// Mitsubishi GX Works2 project: questão_7   PLC: Q03UDV
// LRI_2023

PROGRAM MAIN
VAR
  yo : INT;
  TS0 : BOOL;
  RT0 : BOOL;
END_VAR
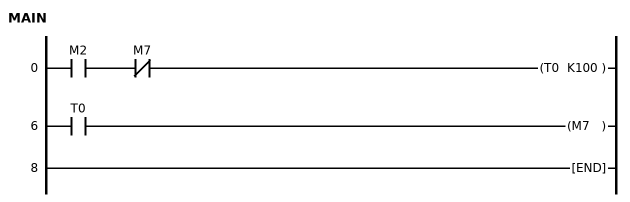
0     LD      M2
      ANI     M7
      OUT     T0 K100
6     LD      T0
      OUT     M7
8     END
END_PROGRAM
